		MoveL Tr_meulage_P550,[50,500,0,0],z0,Tool \wobj:=Wobj_Part_0;
		MoveL Tr_meulage_P551,[50,500,0,0],z0,Tool \wobj:=Wobj_Part_0;
		MoveL Tr_meulage_P552,[50,500,0,0],z0,Tool \wobj:=Wobj_Part_0;
		MoveL Tr_meulage_P553,[50,500,0,0],z0,Tool \wobj:=Wobj_Part_0;
		MoveL Tr_meulage_P554,[50,500,0,0],z0,Tool \wobj:=Wobj_Part_0;
		MoveL Tr_meulage_P555,[50,500,0,0],z0,Tool \wobj:=Wobj_Part_0;
		MoveL Tr_meulage_P556,[50,500,0,0],z0,Tool \wobj:=Wobj_Part_0;
		MoveL Tr_meulage_P557,[50,500,0,0],z0,Tool \wobj:=Wobj_Part_0;
		MoveL Tr_meulage_P558,[50,500,0,0],z0,Tool \wobj:=Wobj_Part_0;
		MoveL Tr_meulage_P559,[50,500,0,0],z0,Tool \wobj:=Wobj_Part_0;
		MoveL Tr_meulage_P560,[50,500,0,0],z0,Tool \wobj:=Wobj_Part_0;
		MoveL Tr_meulage_P561,[50,500,0,0],z0,Tool \wobj:=Wobj_Part_0;
		MoveL Tr_meulage_P562,[50,500,0,0],z0,Tool \wobj:=Wobj_Part_0;
		MoveL Tr_meulage_P563,[50,500,0,0],z0,Tool \wobj:=Wobj_Part_0;
		MoveL Tr_meulage_P564,[50,500,0,0],z0,Tool \wobj:=Wobj_Part_0;
		MoveL Tr_meulage_P565,[50,500,0,0],z0,Tool \wobj:=Wobj_Part_0;
		MoveL Tr_meulage_P566,[50,500,0,0],z0,Tool \wobj:=Wobj_Part_0;
		MoveL Tr_meulage_P567,[50,500,0,0],z0,Tool \wobj:=Wobj_Part_0;
		MoveL Tr_meulage_P568,[50,500,0,0],z0,Tool \wobj:=Wobj_Part_0;
		MoveL Tr_meulage_P569,[50,500,0,0],z0,Tool \wobj:=Wobj_Part_0;
		MoveL Tr_meulage_P570,[50,500,0,0],z0,Tool \wobj:=Wobj_Part_0;
		MoveL Tr_meulage_P571,[50,500,0,0],z0,Tool \wobj:=Wobj_Part_0;
		MoveL Tr_meulage_P572,[50,500,0,0],z0,Tool \wobj:=Wobj_Part_0;
		MoveL Tr_meulage_P573,[50,500,0,0],z0,Tool \wobj:=Wobj_Part_0;
		MoveL Tr_meulage_P574,[50,500,0,0],z0,Tool \wobj:=Wobj_Part_0;
		MoveL Tr_meulage_P575,[50,500,0,0],z0,Tool \wobj:=Wobj_Part_0;
		MoveL Tr_meulage_P576,[50,500,0,0],z0,Tool \wobj:=Wobj_Part_0;
		MoveL Tr_meulage_P577,[50,500,0,0],z0,Tool \wobj:=Wobj_Part_0;
		MoveL Tr_meulage_P578,[50,500,0,0],z0,Tool \wobj:=Wobj_Part_0;
		MoveL Tr_meulage_P579,[50,500,0,0],z0,Tool \wobj:=Wobj_Part_0;
		MoveL Tr_meulage_P580,[50,500,0,0],z0,Tool \wobj:=Wobj_Part_0;
		MoveL Tr_meulage_P581,[50,500,0,0],z0,Tool \wobj:=Wobj_Part_0;
		MoveL Tr_meulage_P582,[50,500,0,0],z0,Tool \wobj:=Wobj_Part_0;
		MoveL Tr_meulage_P583,[50,500,0,0],z0,Tool \wobj:=Wobj_Part_0;
		MoveL Tr_meulage_P584,[50,500,0,0],z0,Tool \wobj:=Wobj_Part_0;
		MoveL Tr_meulage_P585,[50,500,0,0],z0,Tool \wobj:=Wobj_Part_0;
		MoveL Tr_meulage_P586,[50,500,0,0],z0,Tool \wobj:=Wobj_Part_0;
		MoveL Tr_meulage_P587,[50,500,0,0],z0,Tool \wobj:=Wobj_Part_0;
		MoveL Tr_meulage_P588,[50,500,0,0],z0,Tool \wobj:=Wobj_Part_0;
		MoveL Tr_meulage_P589,[50,500,0,0],z0,Tool \wobj:=Wobj_Part_0;
		MoveL Tr_meulage_P590,[50,500,0,0],z0,Tool \wobj:=Wobj_Part_0;
		MoveL Tr_meulage_P591,[50,500,0,0],z0,Tool \wobj:=Wobj_Part_0;
		MoveL Tr_meulage_P592,[50,500,0,0],z0,Tool \wobj:=Wobj_Part_0;
		MoveL Tr_meulage_P593,[50,500,0,0],z0,Tool \wobj:=Wobj_Part_0;
		MoveL Tr_meulage_P594,[50,500,0,0],z0,Tool \wobj:=Wobj_Part_0;
		MoveL Tr_meulage_P595,[50,500,0,0],z0,Tool \wobj:=Wobj_Part_0;
		MoveL Tr_meulage_P596,[50,500,0,0],z0,Tool \wobj:=Wobj_Part_0;
		MoveL Tr_meulage_P597,[50,500,0,0],z0,Tool \wobj:=Wobj_Part_0;
		MoveL Tr_meulage_P598,[50,500,0,0],z0,Tool \wobj:=Wobj_Part_0;
		MoveL Tr_meulage_P599,[50,500,0,0],z0,Tool \wobj:=Wobj_Part_0;
		MoveL Tr_meulage_P600,[50,500,0,0],z0,Tool \wobj:=Wobj_Part_0;
		MoveL Tr_meulage_P601,[50,500,0,0],z0,Tool \wobj:=Wobj_Part_0;
		MoveL Tr_meulage_P602,[50,500,0,0],z0,Tool \wobj:=Wobj_Part_0;
		MoveL Tr_meulage_P603,[50,500,0,0],z0,Tool \wobj:=Wobj_Part_0;
		MoveL Tr_meulage_P604,[50,500,0,0],z0,Tool \wobj:=Wobj_Part_0;
		MoveL Tr_meulage_P605,[50,500,0,0],z0,Tool \wobj:=Wobj_Part_0;
		MoveL Tr_meulage_P606,[50,500,0,0],z0,Tool \wobj:=Wobj_Part_0;
		MoveL Tr_meulage_P607,[50,500,0,0],z0,Tool \wobj:=Wobj_Part_0;
		MoveL Tr_meulage_P608,[50,500,0,0],z0,Tool \wobj:=Wobj_Part_0;
		MoveL Tr_meulage_P609,[50,500,0,0],z0,Tool \wobj:=Wobj_Part_0;
		MoveL Tr_meulage_P610,[50,500,0,0],z0,Tool \wobj:=Wobj_Part_0;
		MoveL Tr_meulage_P611,[50,500,0,0],z0,Tool \wobj:=Wobj_Part_0;
		MoveL Tr_meulage_P612,[50,500,0,0],z0,Tool \wobj:=Wobj_Part_0;
		MoveL Tr_meulage_P613,[50,500,0,0],z0,Tool \wobj:=Wobj_Part_0;
		MoveL Tr_meulage_P614,[50,500,0,0],z0,Tool \wobj:=Wobj_Part_0;
		MoveL Tr_meulage_P615,[50,500,0,0],z0,Tool \wobj:=Wobj_Part_0;
		MoveL Tr_meulage_P616,[50,500,0,0],z0,Tool \wobj:=Wobj_Part_0;
		MoveL Tr_meulage_P617,[50,500,0,0],z0,Tool \wobj:=Wobj_Part_0;
		MoveL Tr_meulage_P618,[50,500,0,0],z0,Tool \wobj:=Wobj_Part_0;
		MoveL Tr_meulage_P619,[50,500,0,0],z0,Tool \wobj:=Wobj_Part_0;
		MoveL Tr_meulage_P620,[50,500,0,0],z0,Tool \wobj:=Wobj_Part_0;
		MoveL Tr_meulage_P621,[50,500,0,0],z0,Tool \wobj:=Wobj_Part_0;
		MoveL Tr_meulage_P622,[50,500,0,0],z0,Tool \wobj:=Wobj_Part_0;
		MoveL Tr_meulage_P623,[50,500,0,0],z0,Tool \wobj:=Wobj_Part_0;
		MoveL Tr_meulage_P624,[50,500,0,0],z0,Tool \wobj:=Wobj_Part_0;
		MoveL Tr_meulage_P625,[50,500,0,0],z0,Tool \wobj:=Wobj_Part_0;
		MoveL Tr_meulage_P626,[50,500,0,0],z0,Tool \wobj:=Wobj_Part_0;
		MoveL Tr_meulage_P627,[50,500,0,0],z0,Tool \wobj:=Wobj_Part_0;
		MoveL Tr_meulage_P628,[50,500,0,0],z0,Tool \wobj:=Wobj_Part_0;
		MoveL Tr_meulage_P629,[50,500,0,0],z0,Tool \wobj:=Wobj_Part_0;
		MoveL Tr_meulage_P630,[50,500,0,0],z0,Tool \wobj:=Wobj_Part_0;
		MoveL Tr_meulage_P631,[50,500,0,0],z0,Tool \wobj:=Wobj_Part_0;
		MoveL Tr_meulage_P632,[50,500,0,0],z0,Tool \wobj:=Wobj_Part_0;
		MoveL Tr_meulage_P633,[50,500,0,0],z0,Tool \wobj:=Wobj_Part_0;
		MoveL Tr_meulage_P634,[50,500,0,0],z0,Tool \wobj:=Wobj_Part_0;
		MoveL Tr_meulage_P635,[50,500,0,0],z0,Tool \wobj:=Wobj_Part_0;
		MoveL Tr_meulage_P636,[50,500,0,0],z0,Tool \wobj:=Wobj_Part_0;
		MoveL Tr_meulage_P637,[50,500,0,0],z0,Tool \wobj:=Wobj_Part_0;
		MoveL Tr_meulage_P638,[50,500,0,0],z0,Tool \wobj:=Wobj_Part_0;
		MoveL Tr_meulage_P639,[50,500,0,0],z0,Tool \wobj:=Wobj_Part_0;
		MoveL Tr_meulage_P640,[50,500,0,0],z0,Tool \wobj:=Wobj_Part_0;
		MoveL Tr_meulage_P641,[50,500,0,0],z0,Tool \wobj:=Wobj_Part_0;
		MoveL Tr_meulage_P642,[50,500,0,0],z0,Tool \wobj:=Wobj_Part_0;
		MoveL Tr_meulage_P643,[50,500,0,0],z0,Tool \wobj:=Wobj_Part_0;
		MoveL Tr_meulage_P644,[50,500,0,0],z0,Tool \wobj:=Wobj_Part_0;
		MoveL Tr_meulage_P645,[50,500,0,0],z0,Tool \wobj:=Wobj_Part_0;
		MoveL Tr_meulage_P646,[50,500,0,0],z0,Tool \wobj:=Wobj_Part_0;
		MoveL Tr_meulage_P647,[50,500,0,0],z0,Tool \wobj:=Wobj_Part_0;
		MoveL Tr_meulage_P648,[50,500,0,0],z0,Tool \wobj:=Wobj_Part_0;
		MoveL Tr_meulage_P649,[50,500,0,0],z0,Tool \wobj:=Wobj_Part_0;
		MoveL Tr_meulage_P650,[50,500,0,0],z0,Tool \wobj:=Wobj_Part_0;
		MoveL Tr_meulage_P651,[50,500,0,0],z0,Tool \wobj:=Wobj_Part_0;
		MoveL Tr_meulage_P652,[50,500,0,0],z0,Tool \wobj:=Wobj_Part_0;
		MoveL Tr_meulage_P653,[50,500,0,0],z0,Tool \wobj:=Wobj_Part_0;
		MoveL Tr_meulage_P654,[50,500,0,0],z0,Tool \wobj:=Wobj_Part_0;
		MoveL Tr_meulage_P655,[50,500,0,0],z0,Tool \wobj:=Wobj_Part_0;
		MoveL Tr_meulage_P656,[50,500,0,0],z0,Tool \wobj:=Wobj_Part_0;
		MoveL Tr_meulage_P657,[50,500,0,0],z0,Tool \wobj:=Wobj_Part_0;
		MoveL Tr_meulage_P658,[50,500,0,0],z0,Tool \wobj:=Wobj_Part_0;
		MoveL Tr_meulage_P659,[50,500,0,0],z0,Tool \wobj:=Wobj_Part_0;
		MoveL Tr_meulage_P660,[50,500,0,0],z0,Tool \wobj:=Wobj_Part_0;
		MoveL Tr_meulage_P661,[50,500,0,0],z0,Tool \wobj:=Wobj_Part_0;
		MoveL Tr_meulage_P662,[50,500,0,0],z0,Tool \wobj:=Wobj_Part_0;
		MoveL Tr_meulage_P663,[50,500,0,0],z0,Tool \wobj:=Wobj_Part_0;
		MoveL Tr_meulage_P664,[50,500,0,0],z0,Tool \wobj:=Wobj_Part_0;
		MoveL Tr_meulage_P665,[50,500,0,0],z0,Tool \wobj:=Wobj_Part_0;
		MoveL Tr_meulage_P666,[50,500,0,0],z0,Tool \wobj:=Wobj_Part_0;
		MoveL Tr_meulage_P667,[50,500,0,0],z0,Tool \wobj:=Wobj_Part_0;
		MoveL Tr_meulage_P668,[50,500,0,0],z0,Tool \wobj:=Wobj_Part_0;
		MoveL Tr_meulage_P669,[50,500,0,0],z0,Tool \wobj:=Wobj_Part_0;
		MoveL Tr_meulage_P670,[50,500,0,0],z0,Tool \wobj:=Wobj_Part_0;
		MoveL Tr_meulage_P671,[50,500,0,0],z0,Tool \wobj:=Wobj_Part_0;
		MoveL Tr_meulage_P672,[50,500,0,0],z0,Tool \wobj:=Wobj_Part_0;
		MoveL Tr_meulage_P673,[50,500,0,0],z0,Tool \wobj:=Wobj_Part_0;
		MoveL Tr_meulage_P674,[50,500,0,0],z0,Tool \wobj:=Wobj_Part_0;
		MoveL Tr_meulage_P675,[50,500,0,0],z0,Tool \wobj:=Wobj_Part_0;
		MoveL Tr_meulage_P676,[50,500,0,0],z0,Tool \wobj:=Wobj_Part_0;
		MoveL Tr_meulage_P677,[50,500,0,0],z0,Tool \wobj:=Wobj_Part_0;
		MoveL Tr_meulage_P678,[50,500,0,0],z0,Tool \wobj:=Wobj_Part_0;
		MoveL Tr_meulage_P679,[50,500,0,0],z0,Tool \wobj:=Wobj_Part_0;
		MoveL Tr_meulage_P680,[50,500,0,0],z0,Tool \wobj:=Wobj_Part_0;
		MoveL Tr_meulage_P681,[50,500,0,0],z0,Tool \wobj:=Wobj_Part_0;
		MoveL Tr_meulage_P682,[50,500,0,0],z0,Tool \wobj:=Wobj_Part_0;
		MoveL Tr_meulage_P683,[50,500,0,0],z0,Tool \wobj:=Wobj_Part_0;
		MoveL Tr_meulage_P684,[50,500,0,0],z0,Tool \wobj:=Wobj_Part_0;
		MoveL Tr_meulage_P685,[50,500,0,0],z0,Tool \wobj:=Wobj_Part_0;
		MoveL Tr_meulage_P686,[50,500,0,0],z0,Tool \wobj:=Wobj_Part_0;
		MoveL Tr_meulage_P687,[50,500,0,0],z0,Tool \wobj:=Wobj_Part_0;
		MoveL Tr_meulage_P688,[50,500,0,0],z0,Tool \wobj:=Wobj_Part_0;
		MoveL Tr_meulage_P689,[50,500,0,0],z0,Tool \wobj:=Wobj_Part_0;
		MoveL Tr_meulage_P690,[50,500,0,0],z0,Tool \wobj:=Wobj_Part_0;
		MoveL Tr_meulage_P691,[50,500,0,0],z0,Tool \wobj:=Wobj_Part_0;
		MoveL Tr_meulage_P692,[50,500,0,0],z0,Tool \wobj:=Wobj_Part_0;
		MoveL Tr_meulage_P693,[50,500,0,0],z0,Tool \wobj:=Wobj_Part_0;
		MoveJ Tr_meulage_degg1,V500,Z0,Tool,\Wobj:=Wobj_Part_0;
		MoveJ Tr_meulage_degg2,V2000,Z100,Tool,\Wobj:=Wobj_Part_0;
	ENDPROC
	 PROC P3_MAIN()
		Tr_pick;
		Tr_Cut;
		Tr_meulage;
	ENDPROC
ENDMODULE
